# EPICS IOC start-up script: acalcout/comp.iocsh
require calc
dbLoadRecords("comp_array.db")
